{attribute addProperty BoxType "EK1100-0000-0018"}
{attribute addProperty Id "Beckhoff_EPP3xxxEK1122Beckhoff_EPP3xxxEK1122_936585F97642955.25"}
{attribute addProperty CRC "1525990897"}
{attribute addProperty SizeInBites "7642"}
{attribute addProperty SizeInBytes "955.25"}
TYPE Beckhoff_EPP3xxx_5AF4C5F1 EXTENDS EK1100_179A0949 :
STRUCT
	{attribute addProperty Name "Beckhoff_EPP3xxxEK1122"}
	Beckhoff_EPP3xxxEK1122 : Beckhoff_EPP3xxxEK1122_936585F9;
END_STRUCT
END_TYPE

(* stored: Version 1.2.0.0, ProductVersion 3.1.4024.9
   DUT Beckhoff_EPP3xxx_5AF4C5F1: Id {e3aeb75c-6322-4c63-a8b0-3c2e59198507} *)
